// TwinCAT 3 PLC project PlcProjekt
// ProgramVersion: 3.1.4022.1
// libraries:
//   Tc2_Standard, * (Beckhoff Automation GmbH)
//   Tc2_System, * (Beckhoff Automation GmbH)
//   Tc2_Utilities, * (Beckhoff Automation GmbH)
//   Tc3_Module, * (Beckhoff Automation GmbH)
// project tree:
//   GVLs/ SimDI.TcGVL (not stored), SimDA.TcGVL (not stored), DigInput.TcGVL (not stored), DigOutput.TcGVL (not stored), AnalogInput.TcGVL, AnalogOutput.TcGVL (not stored), Blinker.TcGVL, VersionsInfo.TcGVL (not stored)
//   / PlcTask.TcTTO (not stored)
//   POUs/ MAIN.TcPOU (not stored), DeleteMe.TcPOU
//   POUs/Privat/ AlleBitSetzen.TcPOU (not stored), BitLesen.TcPOU, DatenRangieren.TcPOU (not stored), SystemFunktionen.TcPOU (not stored)

// ---- GVLs/AnalogInput.TcGVL
{attribute 'qualified_only'}
VAR_GLOBAL
 AI: ARRAY[0..1023] OF BYTE;
END_VAR

// ---- GVLs/Blinker.TcGVL
{attribute 'qualified_only'}
VAR_GLOBAL
	Clock_1Hz:BOOL;
	Clock_1_25Hz:BOOL;
END_VAR

// ---- POUs/Privat/BitLesen.TcPOU
FUNCTION BitLesen : BOOL
VAR_INPUT
Eingang: BYTE;
	Position: BYTE;
END_VAR
VAR
	Bitmuster: BYTE;
END_VAR

Bitmuster := SHL(1, Position);
IF ((Eingang AND Bitmuster) = Bitmuster) THEN
	BitLesen := TRUE;
ELSE		
	BitLesen:= FALSE;	
END_IF;

END_FUNCTION

// ---- POUs/DeleteMe.TcPOU
FUNCTION_BLOCK DeleteMe
VAR_INPUT
END_VAR
VAR_OUTPUT
END_VAR
VAR
	SchrittTransportwagen: INT;
	BeladenAbwarten: TON;
END_VAR

(*  *********************************************************** *)
(*  LAP 2010/2 Transportwagen                                   *)
(*  *********************************************************** *)

IF (NOT SimDI.F1) OR (NOT SimDI.S2) THEN
    SchrittTransportwagen := 100;
END_IF;

CASE SchrittTransportwagen OF
    0:  // Transportwagen steht links (Punkt A)
        SimDA.P1 := FALSE;
        SimDA.Q1 := FALSE;
        SimDA.Q2 := FALSE;
        BeladenAbwarten(IN := FALSE, PT := T#7S); // Timer sind halt so
        IF SimDI.S1 THEN SchrittTransportwagen := 1; END_IF;
        
    1:  // Transportwagen fährt nach rechts (Punkt B)
        SimDA.P1 := FALSE;
        SimDA.Q1 := FALSE;
        SimDA.Q2 := TRUE;
        IF SimDI.B2 THEN SchrittTransportwagen := 2; END_IF;
        
    2: // Transportwagen wartet 7 Sekunden
        SimDA.Q1 := FALSE;
        SimDA.Q2 := FALSE;
        BeladenAbwarten(IN := TRUE, PT := T#7S);
        IF BeladenAbwarten.Q THEN SchrittTransportwagen := 3; END_IF;
        
    3: // Transportwagen fährt zurück links (Punkt A)
        SimDA.P1 := FALSE;
        SimDA.Q1 := TRUE;
        SimDA.Q2 := FALSE;
        IF SimDI.B1 THEN SchrittTransportwagen := 0; END_IF;
        
    100: // Störung aktiv
        SimDA.P1 := (NOT SimDI.F1) OR (NOT SimDI.S2) OR Blinker.Clock_1Hz;
        SimDA.Q1 := FALSE;
        SimDA.Q2 := FALSE;
        IF SimDI.F1 AND SimDI.S2 AND SimDI.S3 THEN SchrittTransportwagen := 3; END_IF;
        
        
    ELSE  // Unbekannter Schritt --> auf was sicheres wechseln
        SchrittTransportwagen := 0;
END_CASE;

END_FUNCTION_BLOCK
